TYPE Warmtepomp_Signalen :
STRUCT
	laagtarief			AT %Q*	: BOOL;
	piekvermogen_uit	AT %Q*	: BOOL;
END_STRUCT
END_TYPE

(* stored: Version 1.1.0.1, ProductVersion 3.1.4024.12
   DUT Warmtepomp_Signalen: Id {2eec57b6-34ab-431a-a0a9-2dbb8aa72f5a} *)
